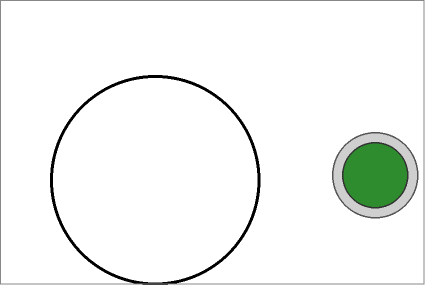
VISUALIZATION VISU_Run_1  // 425x285
    Ellipse (50,75 210x210), "RUN"
        OnMouseDown: execute { GVL.bRun := TRUE; }
        OnMouseUp: execute { GVL.bRun := FALSE; }
    Lamp1 (325,125 100x100), variable: GVL.bRunLamp, style: Lamp-Lamp1-Green
END_VISUALIZATION

(* stored: Version 1.1.0.1
   Visu VISU_Run_1: Id {1bfd8d9d-5e51-47a8-abd4-c1424dfb262a} *)
